FUNCTION_BLOCK FB_SignalGen
VAR_INPUT
END_VAR
VAR_OUTPUT
END_VAR
VAR
END_VAR

END_FUNCTION_BLOCK

(* stored: Version 1.1.0.1, ProductVersion 3.1.4024.12
   POU FB_SignalGen: Id {9e442db7-209c-4d8a-90b5-bb041717cfa9}, SpecialFunc None *)
